ABB RobotStudio station: Entregable2.rspag

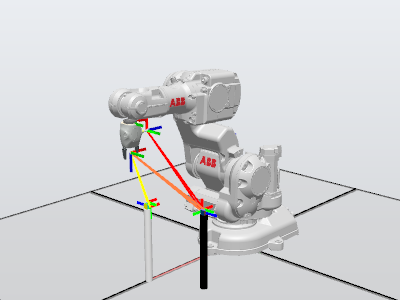
--- station ---
Station Entregable2 (saved by RobotStudio 23.4.10609.1)
Controller Controlador1
  mechanical unit ROB_1: IRB140_6_81_C_03, 6 joints, base frame (0, 0, 0) mm
Layout (positions relative to the parent item):
  - IRB140_6_81_C_03 [mechanism, from %ABB.RobotStudio.Models.IRB140%\IRB140_6_81_C_G_03.rslib] at (0, 0, 0) mm; joint values [-0.0324, 0.3433, -0.3913, 0, 1.6142, 0] (rad or m)
  - Smart_Gripper_Servo_One_Vacuum_Fingers [mechanism, from %ABB.RobotStudio.Models.SmartGripper%\ABB_Smart_Gripper_Servo_One_Vacuum_Fingers.rslib] at (570.72, -18.51, 644.27) mm, rotated rx 180 ry 0.27 rz 178.14 deg; joint values [0.025] (rad or m)
  - Cubo1 [part] at (0, -10, 0) mm, size 20 x 20 x 20 mm
  - Pedestal [part] at (0, -10, 0) mm, size 30 x 30 x 300 mm
  - Cubo2 [part] at (400, 510, 820) mm, rotated rx 49.48 ry 90 rz -40.52 deg, size 20 x 20 x 20 mm
  - Pedestal_2 [part] at (-100, 190, 0) mm, size 30 x 30 x 300 mm
Attachment: Smart_Gripper_Servo_One_Vacuum_Fingers is attached to IRB140_6_81_C_03 / Link6
EventTableEntry 1184: ActivationMode=2, Cyclic=false, Group=, Trigger=DO_Pinza 1185, Actions=[EventTableActionMechanicalPose 1186, EventTableActionDetach 1187], Comment=
EventTableTriggerIO 1185: Operator=0, IOValue=[0], IRC5Controller=? -1, SignalSource=Controlador1 1194
EventTableActionMechanicalPose 1186: VirtualSignal=, Mechanism=Smart_Gripper_Servo_One_Vacuum_Fingers 2274, ToPoseName=PinzaAbierta, VirtualSignalValue=[1]
EventTableActionDetach 1187: AttachmentParent=Smart_Gripper_Servo_One_Vacuum_Fingers 2274, AttachmentChild=? -1
EventTableEntry 1188: ActivationMode=2, Cyclic=false, Group=, Trigger=DO_Pinza 1189, Actions=[EventTableActionMechanicalPose 1190, EventTableActionAttach 1191], Comment=
EventTableTriggerIO 1189: Operator=0, IOValue=[1], IRC5Controller=? -1, SignalSource=Controlador1 1194
EventTableActionMechanicalPose 1190: VirtualSignal=, Mechanism=Smart_Gripper_Servo_One_Vacuum_Fingers 2274, ToPoseName=PinzaCerrada, VirtualSignalValue=[1]
EventTableActionAttach 1191: MountObject=false, FlangeIndext=0, FindNearest=true, AttachmentParent=Smart_Gripper_Servo_One_Vacuum_Fingers 2274, AttachmentChild=? -1, Offset=[X=1, Y=0, Z=0, W=0, X=0, Y=1, Z=0, W=0, X=0, Y=0, Z=1, W=0, X=0, Y=0, Z=0, W=1]
EventTableTriggerIO 2288: Operator=0, IOValue=[0], IRC5Controller=? -1, SignalSource=Controlador1 1194
EventTableTriggerIO 2289: Operator=0, IOValue=[0], IRC5Controller=? -1, SignalSource=Controlador1 1194
EventTableTriggerIO 2290: Operator=0, IOValue=[0], IRC5Controller=? -1, SignalSource=Controlador1 1194
EventTableTriggerIO 2291: Operator=0, IOValue=[0], IRC5Controller=? -1, SignalSource=Controlador1 1194
EventTableTriggerIO 2292: Operator=0, IOValue=[0], IRC5Controller=? -1, SignalSource=Controlador1 1194
EventTableTriggerIO 2293: Operator=0, IOValue=[0], IRC5Controller=? -1, SignalSource=Controlador1 1194
EventTableTriggerIO 2294: Operator=0, IOValue=[0], IRC5Controller=? -1, SignalSource=Controlador1 1194
EventTableTriggerIO 2295: Operator=0, IOValue=[0], IRC5Controller=? -1, SignalSource=Controlador1 1194
EventTableTriggerIO 2296: Operator=0, IOValue=[0], IRC5Controller=? -1, SignalSource=Controlador1 1194
EventTableTriggerIO 2297: Operator=0, IOValue=[0], IRC5Controller=? -1, SignalSource=Controlador1 1194
EventTableTriggerIO 2298: Operator=0, IOValue=[1], IRC5Controller=? -1, SignalSource=Controlador1 1194
EventTableTriggerIO 2299: Operator=0, IOValue=[1], IRC5Controller=? -1, SignalSource=Controlador1 1194
EventTableTriggerIO 2300: Operator=0, IOValue=[1], IRC5Controller=? -1, SignalSource=Controlador1 1194
EventTableTriggerIO 2301: Operator=0, IOValue=[1], IRC5Controller=? -1, SignalSource=Controlador1 1194
EventTableTriggerIO 2302: Operator=0, IOValue=[1], IRC5Controller=? -1, SignalSource=Controlador1 1194
EventTableTriggerIO 2303: Operator=0, IOValue=[1], IRC5Controller=? -1, SignalSource=Controlador1 1194
EventTableTriggerIO 2304: Operator=0, IOValue=[1], IRC5Controller=? -1, SignalSource=Controlador1 1194
EventTableTriggerIO 2305: Operator=0, IOValue=[1], IRC5Controller=? -1, SignalSource=Controlador1 1194
EventTableTriggerIO 2306: Operator=0, IOValue=[1], IRC5Controller=? -1, SignalSource=Controlador1 1194
EventTableTriggerIO 2307: Operator=0, IOValue=[1], IRC5Controller=? -1, SignalSource=Controlador1 1194
EventTableTriggerIO 2416: Operator=0, IOValue=[0], IRC5Controller=? -1, SignalSource=Controlador1 1194
EventTableTriggerIO 2417: Operator=0, IOValue=[1], IRC5Controller=? -1, SignalSource=Controlador1 1194
EventTableTriggerIO 2422: Operator=0, IOValue=[0], IRC5Controller=? -1, SignalSource=Controlador1 1194
EventTableTriggerIO 2423: Operator=0, IOValue=[0], IRC5Controller=? -1, SignalSource=Controlador1 1194
EventTableTriggerIO 2424: Operator=0, IOValue=[0], IRC5Controller=? -1, SignalSource=Controlador1 1194
EventTableTriggerIO 2425: Operator=0, IOValue=[0], IRC5Controller=? -1, SignalSource=Controlador1 1194
EventTableTriggerIO 2426: Operator=0, IOValue=[0], IRC5Controller=? -1, SignalSource=Controlador1 1194
EventTableTriggerIO 2427: Operator=0, IOValue=[0], IRC5Controller=? -1, SignalSource=Controlador1 1194
EventTableTriggerIO 2428: Operator=0, IOValue=[0], IRC5Controller=? -1, SignalSource=Controlador1 1194
EventTableTriggerIO 2429: Operator=0, IOValue=[0], IRC5Controller=? -1, SignalSource=Controlador1 1194
EventTableTriggerIO 2430: Operator=0, IOValue=[0], IRC5Controller=? -1, SignalSource=Controlador1 1194
EventTableTriggerIO 2431: Operator=0, IOValue=[0], IRC5Controller=? -1, SignalSource=Controlador1 1194
EventTableTriggerIO 2432: Operator=0, IOValue=[1], IRC5Controller=? -1, SignalSource=Controlador1 1194
EventTableTriggerIO 2433: Operator=0, IOValue=[1], IRC5Controller=? -1, SignalSource=Controlador1 1194
EventTableTriggerIO 2434: Operator=0, IOValue=[1], IRC5Controller=? -1, SignalSource=Controlador1 1194
EventTableTriggerIO 2435: Operator=0, IOValue=[1], IRC5Controller=? -1, SignalSource=Controlador1 1194
EventTableTriggerIO 2436: Operator=0, IOValue=[1], IRC5Controller=? -1, SignalSource=Controlador1 1194
EventTableTriggerIO 2437: Operator=0, IOValue=[1], IRC5Controller=? -1, SignalSource=Controlador1 1194
EventTableTriggerIO 2438: Operator=0, IOValue=[1], IRC5Controller=? -1, SignalSource=Controlador1 1194
EventTableTriggerIO 2439: Operator=0, IOValue=[1], IRC5Controller=? -1, SignalSource=Controlador1 1194
EventTableTriggerIO 2440: Operator=0, IOValue=[1], IRC5Controller=? -1, SignalSource=Controlador1 1194
EventTableTriggerIO 2441: Operator=0, IOValue=[1], IRC5Controller=? -1, SignalSource=Controlador1 1194
EventTableEntry 2442: ActivationMode=2, Cyclic=false, Group=, Trigger=DO_Gripper 2443, Actions=[EventTableActionAttach 2444], Comment=
EventTableTriggerIO 2443: Operator=0, IOValue=[1], IRC5Controller=? -1, SignalSource=Controlador1 1194
EventTableActionAttach 2444: MountObject=false, FlangeIndext=0, FindNearest=true, AttachmentParent=Smart_Gripper_Servo_One_Vacuum_Fingers 2274, AttachmentChild=? -1, Offset=[X=1, Y=0, Z=0, W=0, X=0, Y=1, Z=0, W=0, X=0, Y=0, Z=1, W=0, X=0, Y=0, Z=0, W=1]
EventTableTriggerIO 2445: Operator=0, IOValue=[1], IRC5Controller=? -1, SignalSource=Controlador1 1194
EventTableTriggerIO 2446: Operator=0, IOValue=[1], IRC5Controller=? -1, SignalSource=Controlador1 1194
EventTableTriggerIO 2447: Operator=0, IOValue=[1], IRC5Controller=? -1, SignalSource=Controlador1 1194
EventTableTriggerIO 2448: Operator=0, IOValue=[1], IRC5Controller=? -1, SignalSource=Controlador1 1194
EventTableTriggerIO 2449: Operator=0, IOValue=[1], IRC5Controller=? -1, SignalSource=Controlador1 1194
EventTableTriggerIO 2450: Operator=0, IOValue=[1], IRC5Controller=? -1, SignalSource=Controlador1 1194
EventTableTriggerIO 2451: Operator=0, IOValue=[1], IRC5Controller=? -1, SignalSource=Controlador1 1194
EventTableTriggerIO 2452: Operator=0, IOValue=[1], IRC5Controller=? -1, SignalSource=Controlador1 1194
EventTableTriggerIO 2453: Operator=0, IOValue=[1], IRC5Controller=? -1, SignalSource=Controlador1 1194
EventTableTriggerIO 2454: Operator=0, IOValue=[1], IRC5Controller=? -1, SignalSource=Controlador1 1194
EventTableEntry 2455: ActivationMode=2, Cyclic=false, Group=, Trigger=DO_Gripper 2456, Actions=[EventTableActionDetach 2457], Comment=
EventTableTriggerIO 2456: Operator=0, IOValue=[0], IRC5Controller=? -1, SignalSource=Controlador1 1194
EventTableActionDetach 2457: AttachmentParent=Smart_Gripper_Servo_One_Vacuum_Fingers 2274, AttachmentChild=? -1
EventTableTriggerIO 2458: Operator=0, IOValue=[0], IRC5Controller=? -1, SignalSource=Controlador1 1194
EventTableTriggerIO 2459: Operator=0, IOValue=[0], IRC5Controller=? -1, SignalSource=Controlador1 1194
EventTableTriggerIO 2460: Operator=0, IOValue=[0], IRC5Controller=? -1, SignalSource=Controlador1 1194
EventTableTriggerIO 2461: Operator=0, IOValue=[0], IRC5Controller=? -1, SignalSource=Controlador1 1194
EventTableTriggerIO 2462: Operator=0, IOValue=[0], IRC5Controller=? -1, SignalSource=Controlador1 1194
EventTableTriggerIO 2463: Operator=0, IOValue=[0], IRC5Controller=? -1, SignalSource=Controlador1 1194
EventTableTriggerIO 2464: Operator=0, IOValue=[0], IRC5Controller=? -1, SignalSource=Controlador1 1194
EventTableTriggerIO 2465: Operator=0, IOValue=[0], IRC5Controller=? -1, SignalSource=Controlador1 1194
EventTableTriggerIO 2466: Operator=0, IOValue=[0], IRC5Controller=? -1, SignalSource=Controlador1 1194
EventTableTriggerIO 2467: Operator=0, IOValue=[0], IRC5Controller=? -1, SignalSource=Controlador1 1194
EventTableTriggerIO 2554: Operator=0, IOValue=[0], IRC5Controller=? -1, SignalSource=Controlador1 1194
EventTableTriggerIO 2555: Operator=0, IOValue=[0], IRC5Controller=? -1, SignalSource=Controlador1 1194
EventTableTriggerIO 2556: Operator=0, IOValue=[0], IRC5Controller=? -1, SignalSource=Controlador1 1194
EventTableTriggerIO 2557: Operator=0, IOValue=[0], IRC5Controller=? -1, SignalSource=Controlador1 1194
EventTableTriggerIO 2558: Operator=0, IOValue=[0], IRC5Controller=? -1, SignalSource=Controlador1 1194
EventTableTriggerIO 2559: Operator=0, IOValue=[0], IRC5Controller=? -1, SignalSource=Controlador1 1194
EventTableTriggerIO 2560: Operator=0, IOValue=[0], IRC5Controller=? -1, SignalSource=Controlador1 1194
EventTableTriggerIO 2561: Operator=0, IOValue=[0], IRC5Controller=? -1, SignalSource=Controlador1 1194
EventTableTriggerIO 2562: Operator=0, IOValue=[0], IRC5Controller=? -1, SignalSource=Controlador1 1194
EventTableTriggerIO 2563: Operator=0, IOValue=[0], IRC5Controller=? -1, SignalSource=Controlador1 1194
EventTableTriggerIO 2564: Operator=0, IOValue=[0], IRC5Controller=? -1, SignalSource=Controlador1 1194
EventTableTriggerIO 2565: Operator=0, IOValue=[0], IRC5Controller=? -1, SignalSource=Controlador1 1194
EventTableTriggerIO 2566: Operator=0, IOValue=[0], IRC5Controller=? -1, SignalSource=Controlador1 1194
EventTableTriggerIO 2567: Operator=0, IOValue=[0], IRC5Controller=? -1, SignalSource=Controlador1 1194
EventTableTriggerIO 2568: Operator=0, IOValue=[0], IRC5Controller=? -1, SignalSource=Controlador1 1194
EventTableTriggerIO 2569: Operator=0, IOValue=[0], IRC5Controller=? -1, SignalSource=Controlador1 1194
EventTableTriggerIO 2570: Operator=0, IOValue=[0], IRC5Controller=? -1, SignalSource=Controlador1 1194
EventTableTriggerIO 2571: Operator=0, IOValue=[0], IRC5Controller=? -1, SignalSource=Controlador1 1194
EventTableTriggerIO 2572: Operator=0, IOValue=[0], IRC5Controller=? -1, SignalSource=Controlador1 1194
EventTableTriggerIO 2573: Operator=0, IOValue=[0], IRC5Controller=? -1, SignalSource=Controlador1 1194
EventTableTriggerIO 2574: Operator=0, IOValue=[1], IRC5Controller=? -1, SignalSource=Controlador1 1194
EventTableTriggerIO 2575: Operator=0, IOValue=[1], IRC5Controller=? -1, SignalSource=Controlador1 1194
EventTableTriggerIO 2576: Operator=0, IOValue=[1], IRC5Controller=? -1, SignalSource=Controlador1 1194
EventTableTriggerIO 2577: Operator=0, IOValue=[1], IRC5Controller=? -1, SignalSource=Controlador1 1194
EventTableTriggerIO 2578: Operator=0, IOValue=[1], IRC5Controller=? -1, SignalSource=Controlador1 1194
EventTableTriggerIO 2579: Operator=0, IOValue=[1], IRC5Controller=? -1, SignalSource=Controlador1 1194
EventTableTriggerIO 2580: Operator=0, IOValue=[1], IRC5Controller=? -1, SignalSource=Controlador1 1194
EventTableTriggerIO 2581: Operator=0, IOValue=[1], IRC5Controller=? -1, SignalSource=Controlador1 1194
EventTableTriggerIO 2582: Operator=0, IOValue=[1], IRC5Controller=? -1, SignalSource=Controlador1 1194
EventTableTriggerIO 2583: Operator=0, IOValue=[1], IRC5Controller=? -1, SignalSource=Controlador1 1194
EventTableTriggerIO 2584: Operator=0, IOValue=[1], IRC5Controller=? -1, SignalSource=Controlador1 1194
EventTableTriggerIO 2585: Operator=0, IOValue=[1], IRC5Controller=? -1, SignalSource=Controlador1 1194
EventTableTriggerIO 2586: Operator=0, IOValue=[1], IRC5Controller=? -1, SignalSource=Controlador1 1194
EventTableTriggerIO 2587: Operator=0, IOValue=[1], IRC5Controller=? -1, SignalSource=Controlador1 1194
EventTableTriggerIO 2588: Operator=0, IOValue=[1], IRC5Controller=? -1, SignalSource=Controlador1 1194
EventTableTriggerIO 2589: Operator=0, IOValue=[1], IRC5Controller=? -1, SignalSource=Controlador1 1194
EventTableTriggerIO 2590: Operator=0, IOValue=[1], IRC5Controller=? -1, SignalSource=Controlador1 1194
EventTableTriggerIO 2591: Operator=0, IOValue=[1], IRC5Controller=? -1, SignalSource=Controlador1 1194
EventTableTriggerIO 2592: Operator=0, IOValue=[1], IRC5Controller=? -1, SignalSource=Controlador1 1194
EventTableTriggerIO 2593: Operator=0, IOValue=[1], IRC5Controller=? -1, SignalSource=Controlador1 1194
EventTableTriggerIO 2594: Operator=0, IOValue=[1], IRC5Controller=? -1, SignalSource=Controlador1 1194
EventTableTriggerIO 2595: Operator=0, IOValue=[1], IRC5Controller=? -1, SignalSource=Controlador1 1194
EventTableTriggerIO 2596: Operator=0, IOValue=[1], IRC5Controller=? -1, SignalSource=Controlador1 1194
EventTableTriggerIO 2597: Operator=0, IOValue=[1], IRC5Controller=? -1, SignalSource=Controlador1 1194
EventTableTriggerIO 2598: Operator=0, IOValue=[1], IRC5Controller=? -1, SignalSource=Controlador1 1194
EventTableTriggerIO 2599: Operator=0, IOValue=[1], IRC5Controller=? -1, SignalSource=Controlador1 1194
EventTableTriggerIO 2600: Operator=0, IOValue=[1], IRC5Controller=? -1, SignalSource=Controlador1 1194
EventTableTriggerIO 2601: Operator=0, IOValue=[1], IRC5Controller=? -1, SignalSource=Controlador1 1194
EventTableTriggerIO 2602: Operator=0, IOValue=[1], IRC5Controller=? -1, SignalSource=Controlador1 1194
EventTableTriggerIO 2603: Operator=0, IOValue=[1], IRC5Controller=? -1, SignalSource=Controlador1 1194
EventTableTriggerIO 2604: Operator=0, IOValue=[1], IRC5Controller=? -1, SignalSource=Controlador1 1194
EventTableTriggerIO 2605: Operator=0, IOValue=[1], IRC5Controller=? -1, SignalSource=Controlador1 1194
EventTableTriggerIO 2606: Operator=0, IOValue=[1], IRC5Controller=? -1, SignalSource=Controlador1 1194
EventTableTriggerIO 2607: Operator=0, IOValue=[1], IRC5Controller=? -1, SignalSource=Controlador1 1194
EventTableTriggerIO 2608: Operator=0, IOValue=[1], IRC5Controller=? -1, SignalSource=Controlador1 1194
EventTableTriggerIO 2609: Operator=0, IOValue=[1], IRC5Controller=? -1, SignalSource=Controlador1 1194
EventTableTriggerIO 2610: Operator=0, IOValue=[1], IRC5Controller=? -1, SignalSource=Controlador1 1194
EventTableTriggerIO 2611: Operator=0, IOValue=[1], IRC5Controller=? -1, SignalSource=Controlador1 1194
EventTableTriggerIO 2612: Operator=0, IOValue=[1], IRC5Controller=? -1, SignalSource=Controlador1 1194
EventTableTriggerIO 2613: Operator=0, IOValue=[1], IRC5Controller=? -1, SignalSource=Controlador1 1194
EventTableTriggerIO 2614: Operator=0, IOValue=[0], IRC5Controller=? -1, SignalSource=Controlador1 1194
EventTableTriggerIO 2615: Operator=0, IOValue=[0], IRC5Controller=? -1, SignalSource=Controlador1 1194
EventTableTriggerIO 2616: Operator=0, IOValue=[0], IRC5Controller=? -1, SignalSource=Controlador1 1194
EventTableTriggerIO 2617: Operator=0, IOValue=[0], IRC5Controller=? -1, SignalSource=Controlador1 1194
EventTableTriggerIO 2618: Operator=0, IOValue=[0], IRC5Controller=? -1, SignalSource=Controlador1 1194
EventTableTriggerIO 2619: Operator=0, IOValue=[0], IRC5Controller=? -1, SignalSource=Controlador1 1194
EventTableTriggerIO 2620: Operator=0, IOValue=[0], IRC5Controller=? -1, SignalSource=Controlador1 1194
EventTableTriggerIO 2621: Operator=0, IOValue=[0], IRC5Controller=? -1, SignalSource=Controlador1 1194
EventTableTriggerIO 2622: Operator=0, IOValue=[0], IRC5Controller=? -1, SignalSource=Controlador1 1194
EventTableTriggerIO 2623: Operator=0, IOValue=[0], IRC5Controller=? -1, SignalSource=Controlador1 1194
EventTableTriggerIO 2624: Operator=0, IOValue=[0], IRC5Controller=? -1, SignalSource=Controlador1 1194
EventTableTriggerIO 2625: Operator=0, IOValue=[0], IRC5Controller=? -1, SignalSource=Controlador1 1194
EventTableTriggerIO 2626: Operator=0, IOValue=[0], IRC5Controller=? -1, SignalSource=Controlador1 1194
EventTableTriggerIO 2627: Operator=0, IOValue=[0], IRC5Controller=? -1, SignalSource=Controlador1 1194
EventTableTriggerIO 2628: Operator=0, IOValue=[0], IRC5Controller=? -1, SignalSource=Controlador1 1194
EventTableTriggerIO 2629: Operator=0, IOValue=[0], IRC5Controller=? -1, SignalSource=Controlador1 1194
EventTableTriggerIO 2630: Operator=0, IOValue=[0], IRC5Controller=? -1, SignalSource=Controlador1 1194
EventTableTriggerIO 2631: Operator=0, IOValue=[0], IRC5Controller=? -1, SignalSource=Controlador1 1194
EventTableTriggerIO 2632: Operator=0, IOValue=[0], IRC5Controller=? -1, SignalSource=Controlador1 1194
EventTableTriggerIO 2633: Operator=0, IOValue=[0], IRC5Controller=? -1, SignalSource=Controlador1 1194
EventTableTriggerIO 2864: Operator=0, IOValue=[0], IRC5Controller=? -1, SignalSource=Controlador1 1194
EventTableTriggerIO 2865: Operator=0, IOValue=[1], IRC5Controller=? -1, SignalSource=Controlador1 1194
EventTableTriggerIO 2866: Operator=0, IOValue=[1], IRC5Controller=? -1, SignalSource=Controlador1 1194
EventTableTriggerIO 2867: Operator=0, IOValue=[0], IRC5Controller=? -1, SignalSource=Controlador1 1194
Targets, tools, work objects and paths stored in the station and not in the controller backup, written as RAPID:
! task T_ROB1
MODULE CalibData
  PERS tooldata Servo:=[TRUE,[[0,0,114.2],[1,0,0,0]],[0.226,[8.9,12.3,48.7],[1,0,0,0],0.00021,0.00024,0.00009]];
  PERS tooldata VaccumOne:=[TRUE,[[63.5,18.5,37.5],[0.707106781,0,0.707106781,0]],[0.226,[8.9,12.3,48.7],[1,0,0,0],0.00021,0.00024,0.00009]];
ENDMODULE

! task T_ROB1
MODULE Module1
  CONST robtarget Home:=[[571.252569574,-18.524401926,530.068410199],[0.002325969,0.016207414,0.999865945,-0.000037696],[-1,0,-1,0],[9E+09,9E+09,9E+09,9E+09,9E+09,9E+09]];
  CONST robtarget Cubo:=[[510,0,325],[0,0,1,0],[0,0,0,0],[9E+09,9E+09,9E+09,9E+09,9E+09,9E+09]];
  CONST robtarget Cubo_Rot:=[[510,15,310],[0,0,-0.707106781,0.707106781],[0,-1,0,0],[9E+09,9E+09,9E+09,9E+09,9E+09,9E+09]];
  CONST robtarget Cubo2:=[[410,200,320],[0,0,1,0],[0,-2,1,0],[9E+09,9E+09,9E+09,9E+09,9E+09,9E+09]];
  CONST robtarget Home2:=[[508.029559094,2.035499351,606.472129196],[0.705367295,-0.011487024,-0.708656686,-0.011433714],[-1,0,-1,0],[9E+09,9E+09,9E+09,9E+09,9E+09,9E+09]];
  CONST robtarget Cubo2_Rot:=[[410,190,310],[0.5,-0.5,-0.5,-0.5],[0,0,1,0],[9E+09,9E+09,9E+09,9E+09,9E+09,9E+09]];
  PROC Rotar_Cubo_Pinza()
    MoveL Home,v200,fine,Servo\WObj:=wobj0;
    MoveL Cubo,v200,fine,Servo\WObj:=wobj0;
    SetDO DO_Pinza,1;
    WaitTime 1;
    MoveL Home,v200,fine,Servo\WObj:=wobj0;
    MoveL Cubo_Rot,v200,fine,Servo\WObj:=wobj0;
    SetDO DO_Pinza,0;
    WaitTime 1;
    MoveL Home,v200,fine,Servo\WObj:=wobj0;
  ENDPROC
  PROC Rotar_Cubo_Vacio()
    MoveL Home2,v200,fine,VaccumOne\WObj:=wobj0;
    MoveL Cubo2,v200,fine,VaccumOne\WObj:=wobj0;
    SetDO DO_Gripper,1;
    WaitTime 1;
    MoveL Home2,v200,fine,VaccumOne\WObj:=wobj0;
    MoveL Cubo2_Rot,v200,fine,VaccumOne\WObj:=wobj0;
    SetDO DO_Gripper,0;
    WaitTime 1;
    MoveL Home2,v200,fine,VaccumOne\WObj:=wobj0;
  ENDPROC
  PROC Ambas()
    MoveL Home,v200,fine,Servo\WObj:=wobj0;
    MoveL Cubo,v200,fine,Servo\WObj:=wobj0;
    SetDO DO_Pinza,1;
    WaitTime 1;
    MoveL Home,v200,fine,Servo\WObj:=wobj0;
    MoveL Cubo_Rot,v200,fine,Servo\WObj:=wobj0;
    SetDO DO_Pinza,0;
    WaitTime 1;
    MoveL Home,v200,fine,Servo\WObj:=wobj0;
    MoveL Cubo2,v200,fine,VaccumOne\WObj:=wobj0;
    SetDO DO_Gripper,1;
    WaitTime 1;
    MoveL Home,v200,fine,Servo\WObj:=wobj0;
    MoveL Cubo2_Rot,v200,fine,VaccumOne\WObj:=wobj0;
    SetDO DO_Gripper,0;
    WaitTime 1;
    MoveL Home,v200,fine,Servo\WObj:=wobj0;
  ENDPROC
ENDMODULE


--- Controller Data/Controlador1/RAPID/TASK1/PROGMOD/Module1.mod ---
MODULE Module1
    !***********************************************************
    !
    ! M?dulo:  Module1
    !
    ! Descripción:
    !   <Introduzca la descripción aquí>
    !
    ! Autor: Javier
    !
    ! Versión: 1.0
    !
    !***********************************************************


    !***********************************************************
    !
    ! Procedimiento Main
    !
    !   Este es el punto de entrada de su programa
    !
    !***********************************************************
    PROC main()
        !Add your code here
    ENDPROC
ENDMODULE

--- Controller Data/Controlador1/SYSPAR/EIO.cfg ---
EIO:CFG_1.0:6:1::
#
EIO_SIGNAL:

      -Name "DO_Pinza" -SignalType "DO" -Access "All"

      -Name "DO_Gripper" -SignalType "DO" -Access "All"
